FUNCTION_BLOCK EnASConsole
  (* Standard: 61499-2 *)
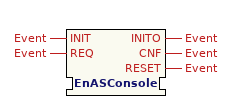
  EVENT_INPUT
    INIT;
    REQ;
  END_EVENT
  EVENT_OUTPUT
    INITO;
    CNF;
    RESET;
  END_EVENT
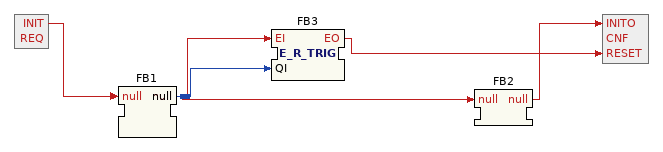
  FBS
    FB1 : ;
    FB2 : ;
    FB3 : E_R_TRIG;
  END_FBS
  EVENT_CONNECTIONS
    INIT TO FB1.null;
    FB1.null TO FB2.null;
    FB2.null TO INITO;
    FB1.null TO FB3.EI;
    FB3.EO TO RESET;
  END_CONNECTIONS
  DATA_CONNECTIONS
    FB1.null TO FB3.QI;
  END_CONNECTIONS
END_FUNCTION_BLOCK
